// TIA Portal V20 export
VAR_GLOBAL   // PLC tag table "Unit1Em3"
   "BA010AZCRPM04.02" AT %Q2012.2 : Bool;   // UNWINDER DANCER FORWARD
   "BA010AZCRPM04.03" AT %Q2012.3 : Bool;   // UNWINDER DANCER BACKWARD
   "BA010AZCRBK05.07" AT %I1016.7 : Bool;   // UNWINDER DANCER SAFETY PIN IDLE POSITION
   "BA010AZCRSP503.02" AT %IW3104 : Int;   // UNWINDER LOADCELL
   "BA010AZCRSP504.00" AT %IW3108 : Int;   // UNWINDER DANCER ENCODER
   "BA010AZCRSP505.00" AT %QW3200 : Int;   // UNWINDER DANCER ELECTRO-PNEUMATIC REGULATOR
END_VAR
VAR_GLOBAL CONSTANT   // user constants
   U1EM3_NO_OF_AXES : USInt := 2;   // Starts with 1. E.g., the value 4 means that 4 axes exist.
   U1EM3_JOB01 : DInt := 1;
   U1EM3_JOB02 : DInt := 2;
   U1EM3_JOB03 : DInt := 3;
   U1EM3_JOB04 : DInt := 4;
   U1EM3_JOB05 : DInt := 5;
   U1EM3_JOB06 : DInt := 6;
   U1EM3_JOB07 : DInt := 7;
   U1EM3_JOB08 : DInt := 8;
   U1EM3_JOB09 : DInt := 9;
   U1EM3_JOB10 : DInt := 10;
   U1EM3_JOB11 : DInt := 11;
   U1EM3_JOB12 : DInt := 12;
   U1EM3_JOB13 : DInt := 13;
   U1EM3_JOB14 : DInt := 14;
   U1EM3_JOB15 : DInt := 15;
   U1EM3_JOB16 : DInt := 16;
   U1EM3_JOB17 : DInt := 17;
   U1EM3_JOB18 : DInt := 18;
   U1EM3_JOB19 : DInt := 19;
   U1EM3_JOB20 : DInt := 20;
   U1EM3_JOB21 : DInt := 21;
   U1EM3_JOB22 : DInt := 22;
   U1EM3_JOB23 : DInt := 23;
   U1EM3_JOB24 : DInt := 24;
   U1EM3_JOB25 : DInt := 25;
   U1EM3_JOB26 : DInt := 26;
   U1EM3_JOB27 : DInt := 27;
   U1EM3_JOB28 : DInt := 28;
   U1EM3_JOB29 : DInt := 29;
   U1EM3_JOB30 : DInt := 30;
   U1EM3_JOB31 : DInt := 31;
   U1EM3_JOB32 : DInt := 32;
   U1EM3_JOB33 : DInt := 33;
   U1EM3_JOB34 : DInt := 34;
   U1EM3_JOB35 : DInt := 35;
   U1EM3_JOB36 : DInt := 36;
   U1EM3_JOB37 : DInt := 37;
   U1EM3_JOB38 : DInt := 38;
   U1EM3_JOB39 : DInt := 39;
   U1EM3_JOB40 : DInt := 40;
   U1EM3_JOB41 : DInt := 41;
   U1EM3_JOB42 : DInt := 42;
   U1EM3_JOB43 : DInt := 43;
   U1EM3_JOB44 : DInt := 44;
   U1EM3_JOB45 : DInt := 45;
   U1EM3_JOB46 : DInt := 46;
   U1EM3_JOB47 : DInt := 47;
   U1EM3_JOB48 : DInt := 48;
   U1EM3_JOB49 : DInt := 49;
   U1EM3_JOB50 : DInt := 50;
END_VAR
